// TIA Portal V20 export
TYPE "LER_typeCommunicationStack"
// stored: Access Published
   STRUCT
      OtherStackToStack { ExternalWritable := 'False'} : "LER_typeCommunicationDataOS2S";
      StackToOtherStack { ExternalWritable := 'False'} : "LER_typeCommunicationDataS2OS";
   END_STRUCT;
END_TYPE
